FUNCTION_BLOCK FB_TP_with_stop
VAR_INPUT
	Start:BOOL;
	Stop:BOOL;
	PT:TIME;
END_VAR
VAR_OUTPUT
	Q:BOOL;
	ET:TIME;
END_VAR
VAR
	R_TRIG_0: R_TRIG;
	TON_0: TON;
	RS_0: RS;
END_VAR

METHOD TP_with_stop
VAR_INPUT
END_VAR
VAR_INST // added by the converter: edge detectors and wires of the graphical bodies
    _w1 : BOOL;
END_VAR
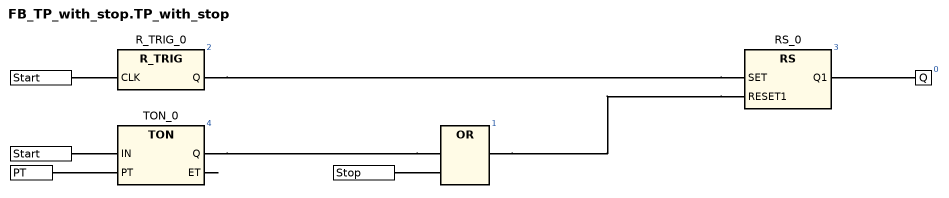
Q := RS_0.Q1;
_w1 := TON_0.Q OR Stop;
R_TRIG_0(CLK := Start); // R_TRIG
RS_0(SET := R_TRIG_0.Q, RESET1 := _w1); // RS
TON_0(IN := Start, PT := PT); // TON
END_METHOD

END_FUNCTION_BLOCK

(* stored: Version 1.1.0.1, ProductVersion 3.1.4024.0
   POU FB_TP_with_stop: Id {3da11ca5-24a2-44a0-8391-220e424d30e1}, SpecialFunc None
   Method TP_with_stop: Id {39a5490e-fdd7-4501-a637-29580e32a887} *)
